FUNCTION_BLOCK FB_Base
VAR_INPUT
    Variable1 : INT;
    Variable2   : DINT;
    Variable3   :REAL;
    Sentence : T_MaxString;
    Conditions : ARRAY[1..6] OF BOOL;
END_VAR
VAR_OUTPUT
END_VAR
VAR
END_VAR

END_FUNCTION_BLOCK

(* stored: Version 1.1.0.1, ProductVersion 3.1.4024.3
   POU FB_Base: Id {a64c0680-a1e5-408a-bb5b-a6bff69faebe}, SpecialFunc None *)
